FUNCTION_BLOCK Valve_mono
VAR_INPUT
	MaxOpenCloseDuration: INT; //(s) Maximum time the valve needs to open or close in seconds
END_VAR
VAR_OUTPUT
	setOpen: BOOL;
END_VAR
VAR_IN_OUT
	Valve: DUT_VALVE;
	I_O: DUT_IO;
END_VAR
VAR
	openingTimer: Tc2_Standard.TON;
	closingTimer: Tc2_Standard.TON;
	fbHmiDut: FB_DUT_HMI; 
	t_reqOpen: BOOL;
	t_reqClose: BOOL;
	t_isOpen: BOOL;
	t_isClosed: BOOL;
	startOpeningTimeOut: BOOL;
	startClosingTimeOut: BOOL;
	t_ioException: BOOL;
	t_stateIoException: BOOL;
	a_setOpen: BOOL;
	a_simIoIsOpen: BOOL;
	a_simIoIsClosed: BOOL;
	t_manualClose: BOOL;
	t_manualOpen: BOOL;
	t_manualReset: BOOL;
END_VAR

{region Input} 
	 
// hmi-open command
IF Valve.Hmi.Open THEN
	t_manualOpen := TRUE;
	Valve.Hmi.Open := FALSE;
END_IF

// hmi-close command
IF Valve.Hmi.Close THEN
	t_manualClose := TRUE;
	Valve.Hmi.Close := FALSE;
END_IF

// manual_reset command
IF Valve.Hmi.Reset THEN
	t_manualReset := TRUE;
	Valve.Hmi.Reset := FALSE;
END_IF 			

Valve.Cs.Open := Valve.Cs.Open AND NOT (Valve.Cs.Close);
{endregion input}

{region manual-auto}
// Convert HMI radioButton input to BOOL's
fbHmiDut(hmiValue_in:= Valve.Hmi);
Valve.Hmi := fbHmiDut.hmiValue_out;

//Set HMI modus overide HMI by CS => (dominant)
Valve.Hmi.DisableAutoManual := Valve.Cs.ManualOn OR Valve.Cs.AutoOn OR Valve.Cs.Interlock;
	 
Valve.Hmi.DisableAutoManual := Valve.Cs.ManualOn OR Valve.Cs.AutoOn;
IF Valve.Cs.ManualOn THEN
	Valve.Hmi.ModeValue := 0;
END_IF

IF Valve.Cs.AutoOn THEN
	Valve.Hmi.ModeValue := 1;
END_IF	  
			   
					
Valve.Hmi.AutoOn := Valve.Hmi.ModeValue = 1;
Valve.Hmi.AutoOff := NOT (Valve.Hmi.AutoOn);
Valve.Hmi.ManualOn := Valve.Hmi.AutoOff;
Valve.Hmi.ManualOff := NOT (Valve.Hmi.ManualOn);

// Set Auto/Manual mode
// CS is Dominant over HMI
Valve.Sts.ManualMode S= (Valve.Cs.Manual OR Valve.Hmi.ManualOn) AND NOT(Valve.Cs.Auto);
Valve.Sts.ManualMode R= (Valve.Cs.Auto OR Valve.Hmi.AutoOn) AND NOT(Valve.Cs.Manual);
Valve.Sts.AutoMode:= NOT(Valve.Sts.ManualMode);

// Get Interlock and simulation from CS and HMI
Valve.Sts.InSimulation := Valve.Cs.Simulation OR Valve.Hmi.Simulation; 
Valve.Sts.Interlock := Valve.Cs.Interlock;	 
		  
{endregion interlock manual auto}
	 
	 
{region internal/temp variables}	 
// determine the actual or required state
t_isClosed := I_O.I_isClosed OR (Valve.Sts.InSimulation AND t_reqClose);
t_isOpen := I_O.I_isOpen OR (Valve.Sts.InSimulation AND t_reqOpen);
t_reqClose := (Valve.Sts.Interlock OR (Valve.Sts.AutoMode AND Valve.Cs.Close) OR (Valve.Sts.ManualMode AND t_manualClose)) AND NOT (t_isClosed);
t_reqOpen := NOT (t_reqClose OR t_isOpen OR Valve.Sts.Interlock) AND ((Valve.Sts.AutoMode AND Valve.Cs.Open) OR (Valve.Sts.ManualMode AND t_manualOpen));
{endregion}

{region control coördination} 
// INIT STS.State zet to CLOSING if UNDEFINED
IF Valve.Sts.State = GVL_VCM.STS_UNDEFINED THEN
	Valve.Sts.State := GVL_VCM.STS_CLOSING;		 
END_IF
// set state
CASE Valve.Sts.State OF
    GVL_VCM.STS_CLOSED: 
	    IF t_reqOpen THEN
    		Valve.Sts.State := GVL_VCM.STS_OPENING;
		END_IF       
    GVL_VCM.STS_OPENING: 
       	IF t_reqClose THEN
   			Valve.Sts.State := GVL_VCM.STS_CLOSING;
		ELSIF t_isOpen THEN
			Valve.Sts.State := GVL_VCM.STS_OPEN;
		END_IF  	  
    GVL_VCM.STS_OPEN: 
        IF t_reqClose THEN
    		Valve.Sts.State := GVL_VCM.STS_Closing;
		END_IF       
    GVL_VCM.STS_CLOSING:
        	IF t_reqOpen THEN
   			Valve.Sts.State := GVL_VCM.STS_OPENING;
		ELSIF t_isClosed THEN
			Valve.Sts.State := GVL_VCM.STS_CLOSED;
		END_IF  	  
END_CASE

Valve.Sts.Closed := Valve.Sts.State = GVL_VCM.STS_CLOSED;
Valve.Sts.Opening := Valve.Sts.State = GVL_VCM.STS_OPENING;
Valve.Sts.Open := Valve.Sts.State = GVL_VCM.STS_OPEN;
Valve.Sts.Closing := Valve.Sts.State = GVL_VCM.STS_CLOSING;
{endregion}

{region set timer guard for opening and closing}
// Don't use the same timer for opening or closing in case opening or closing is called while previous opening or closing action isn't finished yet.
// Can only be done if a 'DirectionChanged' variable is used. 
// opening timeout guard
startOpeningTimeOut S= NOT (Valve.Sts.Interlock) AND Valve.Sts.Opening;
startOpeningTimeOut R= Valve.Sts.Open OR Valve.Sts.Closing;
openingTimer(IN := startOpeningTimeOut, PT:= INT_TO_TIME(MaxOpenCloseDuration * 1000));
// closing timeout guard
startClosingTimeOut S= Valve.Sts.Interlock OR Valve.Sts.Closing;
startClosingTimeOut R= Valve.Sts.Closed OR Valve.Sts.Opening;
closingTimer(IN := startClosingTimeOut, PT:= INT_TO_TIME(MaxOpenCloseDuration * 1000));

{endregion}


IF Valve.Cs.Reset OR t_manualReset THEN
	//reset inAlarm only demand
    Valve.Alm.InAlarm := FALSE;
END_IF

// check if failure(s) (still) exist.
t_stateIoException := (Valve.Sts.Open AND NOT (I_O.I_isOpen)) OR (Valve.Sts.Closed AND NOT (I_O.I_isClosed));
t_ioException := I_O.I_isClosed AND I_O.I_isOpen;	 
Valve.Alm.TimeFailure := openingTimer.Q OR closingTimer.Q; // Set TimeFailure on opening or closing timeOut
Valve.Alm.IsHealthy := I_O.I_isHealthy; // Set GeneralFailure
Valve.Alm.InAlarm := NOT (Valve.Alm.IsHealthy) OR Valve.Alm.TimeFailure OR t_ioException OR t_stateIoException OR Valve.Alm.InAlarm;

{endregion}

{region Actions}

// set/reset output (O_setOpen)
a_setOpen S= (Valve.Sts.Opening OR Valve.Sts.Open); //Warning: Valve is monostable, keep output also open on status: Valve.Sts.Open
a_setOpen R= Valve.Sts.Closing OR Valve.Sts.Interlock OR Valve.Sts.InSimulation;
{endregion}


{region outputs}
// set/reset output (O_setOpen)
I_O.O_setOpen := a_setOpen;

t_manualClose R= TRUE;
t_manualOpen R= TRUE;
t_manualReset R= TRUE;
{endregion}

END_FUNCTION_BLOCK

(* stored: Version 1.1.0.1, ProductVersion 3.1.4024.12
   POU Valve_mono: Id {9c88ac18-dd17-4ae7-b56c-d8d32754d3a0}, SpecialFunc None *)
